{attribute 'qualified_only'}
{attribute 'strict'}
{attribute 'to_string'}
TYPE E_RegelingState :
(
	uit := 0,
	polderpeil,
	debiet
);
END_TYPE

(* stored: Version 1.1.0.1, ProductVersion 3.1.4026.8
   DUT E_RegelingState: Id {9a5da5f4-9fff-4ddd-87be-a4a677063d27} *)
